FUNCTION_BLOCK FB_Syntax_PropertiesFull
VAR
    _fPosition : LREAL;
    _bEnabled  : BOOL;
    _sDevName  : STRING(80);
END_VAR

PROPERTY Enabled : BOOL
GET
Enabled := _bEnabled;
END_GET
SET
_bEnabled := Enabled;
END_SET
END_PROPERTY

PROPERTY Position : LREAL
GET
Position := _fPosition;
END_GET
SET
IF Position >= 0.0 THEN
    _fPosition := Position;
END_IF
END_SET
END_PROPERTY

END_FUNCTION_BLOCK

(* stored: Version 1.1.0.1, ProductVersion 3.1.4024.16
   POU FB_Syntax_PropertiesFull: Id {6a851fec-f539-4349-b078-7a9f80c57bab}, SpecialFunc None
   Property Enabled: Id {edddc1b8-ba0c-4a5c-a814-db1c51387ed5}
   Get Get: Id {c621d76c-7d28-4edb-8721-8a8e09632dee}
   Set Set: Id {37508d12-1ba5-43d2-8c05-5d4337df8d50}
   Property Position: Id {a152f216-7144-461d-9387-da22dcd40d18}
   Get Get: Id {b818b00c-d33f-486e-85c1-1af992d94060}
   Set Set: Id {b7db9a44-aeb5-4e4d-b796-103760e5b07c} *)
